FUNCTION_BLOCK FB_EmonioP3
VAR_INPUT
	sIPAddr : STRING(15);
END_VAR
VAR_OUTPUT
	fPower : REAL; 			//kW
	fVoltage : REAL; 		//V
	fCurrent : REAL; 		//A
	fEnergy : REAL; 		//kWh
	fTemperature : REAL; 	//°C
	fPulse : REAL; 			//m^3
	
	bErrorEM: BOOL;
	bErrorTemp: BOOL;
	bErrorPulse : BOOL;
END_VAR
VAR
	{attribute 'OPC.UA.DA' := '1'}
	sensorState : ST_EmonioP3State;
	
	fbEmonioElectricity : FB_MBReadRegs;
	fbEmonioTemperature : FB_MBReadRegs;
	fbEmonioPulse : FB_MBReadRegs;
	
	//timer to execute modbus fb
	Timer : TON;	
	bStartTimer : BOOL;
	bReadModbus : BOOL;
	
	arrInputRegsElectricity: ARRAY[0..13] OF WORD;			  // buffer for modbus fb electricity values
	arrInputRegsTemperature: ARRAY[0..1] OF WORD;			  // buffer for modbus fb temperature value
	arrInputRegsPulse: ARRAY[0..1] OF WORD;			  // buffer for modbus fb pulse value
	
    nErrIdEM: UDINT;
    nErrIdTemp: UDINT;
	nErrIdPulse: UDINT;
	
	//define arrays to convert from 16-bit word to real values
	PowerArray: ARRAY [0..1] OF WORD;
	VoltageArray: ARRAY [0..1] OF WORD;
	CurrentArray: ARRAY [0..1] OF WORD;
	EnergyArray: ARRAY [0..1] OF WORD;
	TemperatureArray: ARRAY [0..1] OF WORD;
	PulseArray: ARRAY [0..1] OF WORD;
	
	PowerInWatt : REAL; //helper variable to convert from W to kW
END_VAR

//Start and check timer for 2s interval
Timer(IN := bStartTimer,
	PT := T#2S);
bStartTimer := TRUE;
IF Timer.Q THEN
	bReadModbus := TRUE;
	bStartTimer := FALSE;	
END_IF

// Read Emonio via Modbus
fbEmonioElectricity(    
	sIPAddr := sIPAddr,   			//IP adress of the device
	nTCPPort := 502,				//Port number of the target device
	nUnitID := 255,					//Identification number of a serial sub-network device
	nQuantity  := 13,				//Number of input registers (data words) to be read
	nMBAddr := 0,					// Start address of the output registers to be read (word offset)
	cbLength := SIZEOF(arrInputRegsElectricity),
	pDestAddr := ADR(arrInputRegsElectricity),
	bExecute := bReadModbus,         // trigger
	tTimeout  := T#20S,
	bError => bErrorEM,				// Error handling
	nErrId => nErrIdEM				// Error handling 
);

fbEmonioTemperature(    
	sIPAddr := sIPAddr,   			//IP adress of the device
	nTCPPort := 502,				//Port number of the target device
	nUnitID := 255,					//Identification number of a serial sub-network device
	nQuantity  := 2,				//Number of input registers (data words) to be read
	nMBAddr := 500,					// Start address of the output registers to be read (word offset)
	cbLength := SIZEOF(arrInputRegsTemperature),
	pDestAddr := ADR(arrInputRegsTemperature),
	bExecute := bReadModbus,         // trigger
	tTimeout  := T#20S,
	bError => bErrorTemp,				// Error handling
	nErrId => nErrIdTemp				// Error handling 
);

fbEmonioPulse(    
	sIPAddr := sIPAddr,   			//IP adress of the device
	nTCPPort := 502,				//Port number of the target device
	nUnitID := 255,					//Identification number of a serial sub-network device
	nQuantity  := 2,				//Number of input registers (data words) to be read
	nMBAddr := 800,					// Start address of the output registers to be read (word offset)
	cbLength := SIZEOF(arrInputRegsPulse),
	pDestAddr := ADR(arrInputRegsPulse),
	bExecute := bReadModbus,         // trigger
	tTimeout  := T#20S,
	bError => bErrorPulse,				// Error handling
	nErrId => nErrIdPulse				// Error handling 
);

bReadModbus := FALSE;

//create arrays with word outputs
PowerArray[0] := arrInputRegsElectricity[4];
PowerArray[1] := arrInputRegsElectricity[5];
VoltageArray[0] := arrInputRegsElectricity[0];
VoltageArray[1] := arrInputRegsElectricity[1];
CurrentArray[0] := arrInputRegsElectricity[2];
CurrentArray[1] := arrInputRegsElectricity[3];
EnergyArray[0] := arrInputRegsElectricity[12];
EnergyArray[1] := arrInputRegsElectricity[13];
TemperatureArray[0] := arrInputRegsTemperature[0];
TemperatureArray[1] := arrInputRegsTemperature[1];
PulseArray[0] := arrInputRegsPulse[0];
PulseArray[1] := arrInputRegsPulse[1];

//convert word to real values
MEMCPY(ADR(PowerInWatt), ADR(PowerArray), 4);
sensorState.fPower := PowerInWatt/1000;
MEMCPY(ADR(sensorState.fVoltage), ADR(VoltageArray), 4);
MEMCPY(ADR(sensorState.fCurrent), ADR(CurrentArray), 4);
MEMCPY(ADR(sensorState.fEnergy), ADR(EnergyArray), 4);
MEMCPY(ADR(sensorState.fTemperature), ADR(TemperatureArray), 4);
MEMCPY(ADR(sensorState.fPulse), ADR(PulseArray), 4);

//define output variables
fPower := sensorState.fPower;
fVoltage := sensorState.fVoltage;
fCurrent := sensorState.fCurrent;
fEnergy := sensorState.fEnergy;
fTemperature := sensorState.fTemperature;
fPulse := sensorState.fPulse;

END_FUNCTION_BLOCK

(* stored: Version 1.1.0.1, ProductVersion 3.1.4024.10
   POU FB_EmonioP3: Id {c4a1a050-55fe-4479-b0af-783598946749}, SpecialFunc None *)
